INTERFACE I_RpcDynamicConfigBuild

METHOD Build : HRESULT
VAR_INPUT
END_VAR
END_METHOD

END_INTERFACE

(* stored: Version 1.1.0.1, ProductVersion 3.1.4024.12
   Itf I_RpcDynamicConfigBuild: Id {d14865a4-cf7b-43ff-9162-516200461cd5}
   Method Build: Id {3eefaa5b-d67b-489f-9887-46326278cddd} *)
